INTERFACE I_CamBuildSequence EXTENDS I_SequenceTest

END_INTERFACE

(* stored: Version 1.1.0.1, ProductVersion 3.1.4026.19
   Itf I_CamBuildSequence: Id {51efc471-2182-472f-b1fb-387c8e510691} *)
